TYPE ST_GripperRequest :
STRUCT
    eCommand      : E_GripperCommand; // 本次请求的动作
    udiRequestId  : UDINT;            // 每发起一条新命令递增一次
                                      // 功能块只处理新的编号，避免持续重复发送
END_STRUCT
END_TYPE

(* stored: Version 1.1.0.1, ProductVersion 3.1.4026.20
   DUT ST_GripperRequest: Id {b4c9a931-36ae-45b9-ba53-ad25187fa198} *)
